KUKA KRL data list: mhekxdemo.dat

&ACCESS RVP
&PARAM TEMPLATE = C:\KRC\Roboter\Template\vorgabe
&PARAM EDITMASK = *
DEFDAT mhekxdemo
ENDDAT
